PROGRAM LaserMarking_Variable_Selection
VAR
END_VAR

END_PROGRAM

(* stored: Version 1.1.0.1, ProductVersion 3.1.4024.0
   POU LaserMarking_Variable_Selection: Id {6e9c51ea-65b6-4e4f-8cba-cf61000ffbfe}, SpecialFunc None *)
